// TIA Portal V16 export
// export: Created 2021-07-03T21:22:43.7684864Z, ExportSetting WithDefaults, DisplayName Totally Integrated Automation Portal, DisplayVersion V16, DisplayName TIA Portal Version Control Interface, DisplayVersion V16, DisplayName TIA Portal Openness, DisplayVersion V16, DisplayName STEP 7 Professional, DisplayVersion V16, DisplayName STEP 7 Safety, DisplayVersion V16, DisplayName WinCC Professional, DisplayVersion V16
TYPE "118MK2_PlantIF_Cmd_OPC"
// stored: IsFailsafeCompliant false
   STRUCT
      Start_M_PCS : Bool;   // Moves machine to Processing Material State. Feeder is not started.
      Stop_M_PCS : Bool;   // Moves machine to Standby State. Hence also used to exit Display mode.
      Start_Feeding_M_PCS : Bool;   // Starts the vibratory feeder
      Stop_Feeding_M_PCS : Bool;   // Stops the vibratory feeder
      Checker_Cycle_M_PCS : Bool;   // Initiates a Checker Cycle sequence
      Purge_M_PCS : Bool;   // Initiates a material purge sequence
      Acknowledge_Alarm_PCS : Bool;   // Acknowledges asserted alarm/s. Siren is deactivated.
      Reset_Alarm_PCS : Bool;   // Resets asserted alarm/s
      Manual_Req_PCS : Bool;   // Initiates a Mode Request, Toggles between Manual/Auto
      Calibrate_M_PCS : Bool;   // Automatically adjusts the PMT HV setpoints to achieve the desired calibration reference
      Display_M_PCS : Bool;   // Moves machine to Display state where blue and red channel data for all 8 channels is acquired every 250ms
      Save_As_Reference_PCS : Bool;   // Saves the most recent calibration data for both the blue and red channels as the reference curve in the RT Controller non-volatile memory
      Save_Oper_Params_PCS : Bool;   // Saves all operation parameters to NVM on the RT Controller
      Upd_Sys_DateTime_PCS : Bool;   // Issue a System Date and Time Update
      Spare6 : Bool;   // Spare
      Spare7 : Bool;   // Spare
      Clr_LiHist_M_PCS : Bool;   // Clears Accepted, Rejected, Red and Blue-Red Ratio Luminescence Intensity Histograms
      Clr_Profile_M_PCS : Bool;   // Clears ejection, accepted & rejected profiles
      Clr_EjecErrHist_M_PCS : Bool;   // Resets all the data values in the Ejector error histograms to zero
      Clr_EjecResProf_M_PCS : Bool;   // Clears ejector delay response and ejector duration response profiles
      Clr_CCCalData_M_PCS : Bool;   // Clears Blue and Red Checker cycle calibration data profiles
      Spare8 : Bool;   // Spare
      Spare9 : Bool;   // Spare
      Spare10 : Bool;   // Spare
      Spare11 : Bool;   // Spare
      Spare12 : Bool;   // Spare
      Spare13 : Bool;   // Spare
      Spare14 : Bool;   // Spare
      Spare15 : Bool;   // Spare
      Spare16 : Bool;   // Spare
      Spare17 : Bool;   // Spare
      Spare18 : Bool;   // Spare
      Add_New_User_PCS : Bool;   // Adds a new User based Username, password and Access level
      Del_Select_User_PCS : Bool;   // Delete the user specified by the current lookup table pointer, from the cRIO security lookup table
      Logon_User_PCS : Bool;   // Authorise user based on the specified username and password - the cRIO would return the appropriate access level
      LogOff_User_PCS : Bool;   // Log off user – the Access Level of 0 would return after command
      Change_User_Pass_PCS : Bool;   // Change password for currently logged on user as specified in “User password”
      Lookup_User_PCS : Bool;   // Retrieve the Username and Access Level at the specified Sec. Lookup table pntr
      Spare19 : Bool;   // Spare
      Spare20 : Bool;   // Spare
      Start_A_PCS : Bool;   // Sequencer Start
      Stop_A_PCS : Bool;   // Sequencer Stop
      Start_Feeding_A_PCS : Bool;   // Sequencer Feeder Start
      Stop_Feeding_A_PCS : Bool;   // Sequencer Feeder Stop
      Checker_Cycle_A_PCS : Bool;   // Sequencer Checker Cycle Req
      Purge_A_PCS : Bool;   // Sequencer Purge Req
      Spare21 : Bool;   // Spare
      Spare22 : Bool;   // Spare
      User_Name : Array[0..7] of Byte;   // User Name for Authorization/addition on Machine lookup table
      User_Password : Array[0..7] of Byte;   // User Password for Authorization/addition on Machine lookup table
      User_Access_Level : Byte;   // User Access Level for Addintion on Machine Lookup table
      Sec_LookupTable_Pntr : Byte := 16#0;   // Lookup user in security lookup table. Range: 1 to 40. 0 = hidden administrator.
      Save_Recipe : Bool;   // 1 to Save Current Recipe
      Delete_Recipe : Bool;   // 1 to Delete Current Recipe
      Copy_Recipe : Bool;   // 1 to Copy a Recipe
      Spare23 : Bool;   // Spare
      Spare24 : Bool;   // Spare
      Spare25 : Bool;   // Spare
      Spare26 : Bool;   // Spare
      Spare27 : Bool;   // Spare
      Select_Recipe_No : Byte;   // Select Active Recipe
      Dest_Recipe_No : Byte;   // Set the Destination Number to copy to
      Spare28 : Byte;   // Spare
      ScratchPad : "118MK2_RecipeEdit";   // Scratch Pad for Recipe Edits
      Remote_DSInlk_PCS : Bool;   // Status of the D/S int. on either MachPLC-H/W or PlntPLC-S/W 0: Inlk 1: Healthy
      Remote_SpareCMD1_PCS : Bool;   // Spare Remote Commands
      Remote_SpareCMD2_PCS : Bool;   // Spare Remote Commands
      Remote_SpareCMD3_PCS : Bool;   // Spare Remote Commands
      Remote_SpareCMD4_PCS : Bool;   // Spare Remote Commands
      Remote_SpareCMD5_PCS : Bool;   // Spare Remote Commands
      Remote_SpareCMD6_PCS : Bool;   // Spare Remote Commands
      Remote_SpareCMD7_PCS : Bool;   // Spare Remote Commands
      SOC_Authorization : Bool;   // Supervised Operator Control Authorization, 0 = No Auth, 1 = Grant Auth
      SOC_Req_Acknowledge : Bool;   // Spare
      Spare30 : Bool;   // Spare
      Spare31 : Bool;   // Spare
      Spare32 : Bool;   // Spare
      Spare33 : Bool;   // Spare
      Spare34 : Bool;   // Spare
      Spare35 : Bool;   // Spare
      Heartbeat_PCS_MPLC : Byte;   // Receive Comms Heartbeat from Plant PLC
      Spare36 : Byte;   // Spare
      RTC_Update_PCS { S7_SetPoint := 'True'} : "RTC";   // Real Time Clock Update Data
      PCS_Data_Range : Byte;   // Plant data range: 0 (default)= Basic command and statuses; 1=Include messages; 2=Include MAPCOM data
      Spare37 : Byte;   // Spare
      Spare38 : Word;   // Spare
      Spare39 : Word;   // End of Receive Data Structure - 70 Bytes
   END_STRUCT;
END_TYPE
